FUNCTION_BLOCK FB_XPlanar_EM EXTENDS FB_PackML_BaseModule
VAR
    // Sub module definitions here

    // List of sub modules
    ipSubModules_Init : ARRAY[1..Parameters_PackML_Base.MAX_NO_OF_SUBMODULES] OF I_PackML_BaseModule := [];

    // Component definitions here
    XPlanarTable : FB_Component_Xplanar := (Name := 'XPlanarTable');
	
	//Station Components
	Station1	 : FB_DecisionStation	 := (Name := 'DecisionPoint');   //Declaration of a custom station
	Station2	 : FB_SpinStation 		 := (Name := 'RotateStation');
	Station3	 : FB_XPlanarStationBase := (Name := 'InspectStation');  //If no custom processing is needed simply declare an instance of the Station Base fb	 

    // List of Components
    ipComponents_Init : ARRAY[1..Parameters_PackML_Base.MAX_NO_OF_COMPONENTS] OF I_ComponentBase := [XPlanarTable, Station1, Station2, Station3];

    //Helper Vars
	Movers			  : ARRAY[1..Tc3_XPlanarStandard.Params_XPlanar.moverCount] OF FB_XPlanarMover;
	Tracks			  : ARRAY[1..Tc3_XPlanarStandard.Params_XPlanar.maxTrackCount] OF FB_XPlanarTrackSegment;
	
	
	fbinitbasic						: FB_BasicInitialization;
	aLocationOfArea 			: ARRAY[1..4,1..2] OF REAL:=[0,480,960,480,0,0,960,0];
	aManualPos					: ARRAY [1..19,1..2] OF REAL:=[60,420,240,420,420,420,600,420,860,420,60,300,240,300,420,300,600,300,860,300,60,180,240,180,420,180,600,180,860,180, 60,60,310,60,560,60,820,60];	
	
END_VAR

//! @summary This method contains code which will execute when this PackML module is in the <b>Aborting</b> state
METHOD PROTECTED Aborting
VAR
    i               : UDINT;
    SubModulesReady : BOOL := TRUE;
END_VAR

(*! <description> <b>Note:</b> The <i>Abort</i> command should be associated with the fault handing routine of a module. It should not be directly commanded from any user inteface. 

<table> 
	<tr>
		<th> Previous State </th>
		<th> Transition In </th>
		<th> Transition Out </th>
		<th> Next State  </th> 
	</tr>
	<tr>
		<td> <b>ANY</b> </td>
		<td> Abort Command </td> 
		<td> State Complete </td>
		<td> Aborted </td> 
	</tr>
</table>

This method is called as required by <c>StateControl()</c>
</description> 

*)
CASE DescendantSequenceState OF
    0:
        NoStateTasksToComplete  := FALSE;
        DescendantSequenceState := NextStep(DescendantSequenceState);

    10:
        IF XPlanarTable.Abort() THEN
            StateTasksComplete      := TRUE;
            DescendantSequenceState := NextStep(DescendantSequenceState);
        END_IF

    20:
        StateTasksComplete := TRUE;
END_CASE

SUPER^.Aborting();
END_METHOD

//! @summary This method contains code which will execute when this PackML module is in the <b>Clearing</b> state
METHOD PROTECTED Clearing
VAR
    i               : UDINT;
    SubModulesReady : BOOL := TRUE;
END_VAR

(*! <description> <b>Note:</b> The <i>Clear</i> command can also be thought of as a <i>fault reset</i> depite the ambiguity in the naming of the <i>Reset</i> state. 
<table> 
	<tr>
		<th> Previous State </th>
		<th> Transition In </th>
		<th> Transition Out </th>
		<th> Next State  </th> 
	</tr>
	<tr>
		<td> Aborted </td>
		<td> Clear Command </td> 
		<td> State Complete </td>
		<td> Stopped </td> 
	</tr>
</table>
This method is called as required by <c>StateControl()</c>
</description> 

*)
CASE _CurrentMode OF
    E_PMLUnitMode.ePMLUnitMode_Production:
        CASE DescendantSequenceState OF
            0: //Init
                NoStateTasksToComplete  := FALSE;
                XPlanarTable._Error     := FALSE;
				Station1.Reset();
				Station2.Reset();
				Station3.Reset();
			
                DescendantSequenceState := NextStep(DescendantSequenceState);

            10: //Check for Track initialization
                IF NOT XPlanarTable.TracksInitialized THEN
                    DescendantSequenceState := NextMinorStep(DescendantSequenceState);
                ELSE
                    DescendantSequenceState := NextStep(DescendantSequenceState);
                END_IF

            11: //Build Track Segments
                IF XPlanarTable.BuildTracks() THEN
                    IF NOT XPlanarTable.Error THEN
                      DescendantSequenceState := NextStep(DescendantSequenceState);
                    ELSE
                        DescendantSequenceState := 999;
                    END_IF;
                END_IF

            20: //Enable Group
                IF XPlanarTable.EnableGroup() THEN
                    DescendantSequenceState := NextStep(DescendantSequenceState);
                END_IF

            30:
                //Clearing complete
				fbinitbasic(bReset:=TRUE);
                StateTasksComplete := TRUE;
        END_CASE

    E_PMLUnitMode.ePMLUnitMode_Manual:
        ;
END_CASE

SUPER^.Clearing();
END_METHOD

METHOD PROTECTED CreateEvents
VAR_INPUT
END_VAR
// Add your event creation here

// Super call to base
SUPER^.CreateEvents();
END_METHOD

METHOD CyclicLogic
VAR
    i : INT;
    j : UDINT;
END_VAR
IF NOT _InitComplete THEN
    _InitComplete := Initialize();
END_IF

SUPER^.CyclicLogic();

IF _InitComplete THEN
	FOR j := 1 TO MAX_STATION_NUMBER DO
		stStationVis[j].bInit := TRUE;
		stStationVis[j].fPosition_X := stStationPos[j].fpositionX;		
		stStationVis[j].fPosition_Y := stStationPos[j].fpositionY;		
	END_FOR
	FOR j := 1 TO Tc3_XPlanarStandard.Params_XPlanar.moverCount DO
		stMoverVis[j].fPosition_X := Movers[j].std.P_ActPosition.x;		
		stMoverVis[j].fPosition_Y := Movers[j].std.P_ActPosition.y;	
		stMoverVis[j].fPosition_C := Movers[j].std.P_ActPosition.c;			
	END_FOR	
	

END_IF
END_METHOD

//! @summary This method contains code which will execute when this PackML module is in the <b>Execute</b> state
METHOD PROTECTED Execute
VAR
    i : UDINT;
END_VAR
VAR_INST
	InspectSimTimer: TON;
END_VAR
(*! <description> <b>The base implementation of this method is empty. User must override this method to provide functionality.</b>
<table> 
	<tr>
		<th> Previous State </th>
		<th> Transition In </th>
		<th> Transition Out </th>
		<th> Next State  </th> 
	</tr>
	<tr>
		<td> Starting<b>-or-</b>Unholding <b>-or-</b>Unsuspending</td>
		<td> State Complete<i>(Starting<b>-or-</b>Unholding<b>-or-</b>Unsuspending)</i></td> 
		<td> State Complete<b>-or-</b>Hold Command<b>-or-</b>Suspend Command</td>
		<td> Completing<b>-or-</b>Holding<b>-or-</b>Suspending</td>
	</tr>
</table>
This method is called as required by <c>StateControl()</c>
</description> 

*)
CASE _CurrentMode OF
    E_PMLUnitMode.ePMLUnitMode_Production:
        FOR i := 1 TO Params_XPlanar.maxNumStation DO
            ip.Stations[i].Execute();
        END_FOR
	
	//Simulate the "Inspection Done" signal
	InspectSimTimer(IN := ip.Stations[3].StationReady, PT := T#1S);
	ip.Stations[3].StationComplete := InspectSimTimer.Q;
	
    E_PMLUnitMode.ePMLUnitMode_Manual:
        ;
END_CASE
END_METHOD

//! @summary Automatically enables and disables HMI control based on the PackML mode
METHOD PROTECTED HMIPermissions

//! @description This method is called cyclically by <c>CyclicLogic()</c>
//General Mode Based Monitoring and handling of HMI control
CASE _CurrentMode OF
    E_PMLUnitMode.ePMLUnitMode_Production:
        AllowHMIControl(ThisModuleOnly := FALSE);

    E_PMLUnitMode.ePMLUnitMode_Manual:
        AllowHMIControl(ThisModuleOnly := FALSE);

    E_PMLUnitMode.ePMLUnitMode_Maintenance:
        AllowHMIControl(ThisModuleOnly := FALSE);
END_CASE
END_METHOD

//! @summary Basic module initialization logic
METHOD PROTECTED Initialize : BOOL;
VAR
    i                        : UDINT;
    varInfo                  : __SYSTEM.VAR_INFO;
    AllSubUnitsInitialized   : BOOL := TRUE;
    AllComponentsInitialized : BOOL := TRUE;
    tmpMoveDynamics          : ST_MoveDynamics;
    stHaltDynamics           : ST_HaltDynamics;
END_VAR

//! @description This method is called by <c>CyclicLogic()</c> as required
Initialize := FALSE;
CASE DescendantSequenceState OF
	0:
		// Define the interfaces to the different subunits (Must take place before SUPER^.initialize call)
		FOR i := 1 TO SPT_BaseTypes.Parameters_PackML_Base.MAX_NO_OF_SUBMODULES DO
			ipSubModules[i] := ipSubModules_Init[i];
		END_FOR

		FOR i := 1 TO SPT_BaseTypes.Parameters_PackML_Base.MAX_NO_OF_COMPONENTS DO
			ipComponents[i] := ipComponents_Init[i];
		END_FOR

		_LogModeChanges			:= FALSE;
		_LogStateChanges		:= FALSE;
		DescendantSequenceState := DescendantSequenceState + 10;

	10:
		//Set Mover and Track interfaces
		FOR i := 1 TO Tc3_XPlanarStandard.Params_XPlanar.moverCount DO
			Movers[i].MoverIndex := i;
			ip.Movers[i]		  := Movers[i];
		END_FOR

		FOR i := 1 TO Tc3_XPlanarStandard.Params_XPlanar.maxTrackCount DO
			ip.Tracks[i] := Tracks[i];
		END_FOR

		DescendantSequenceState := DescendantSequenceState + 10;

	20:
		//Copy Mode names
		FOR i := 1 TO 3 DO
			ModeNames[i] := F_UnitModeToString(UDINT_TO_DINT(i));
		END_FOR

		DescendantSequenceState := DescendantSequenceState + 10;

	30:
		//Call the Super
		IF SUPER^.Initialize() THEN
			DescendantSequenceState := DescendantSequenceState + 10;
		END_IF

	40:
		IF SetupTrackSegments() THEN
			DescendantSequenceState := DescendantSequenceState + 10;
		END_IF

	50:
		IF SetupStations() THEN
			DescendantSequenceState := DescendantSequenceState + 10;
		END_IF

	60:
		stHaltDynamics.PathXY.fVelocity		:= 500.0;
		stHaltDynamics.PathXY.fAcceleration := 10000.0;
		stHaltDynamics.PathXY.fDeceleration := 10000.0;
		stHaltDynamics.PathXY.fJerk			:= 100000.0;
		stHaltDynamics.AxisX.fVelocity		:= 500.0;
		stHaltDynamics.AxisX.fAcceleration	:= 10000.0;
		stHaltDynamics.AxisX.fDeceleration	:= 10000.0;
		stHaltDynamics.AxisX.fJerk			:= 100000.0;
		stHaltDynamics.AxisY.fVelocity		:= 500.0;
		stHaltDynamics.AxisY.fAcceleration	:= 10000.0;
		stHaltDynamics.AxisY.fDeceleration	:= 10000.0;
		stHaltDynamics.AxisY.fJerk			:= 100000.0;
		stHaltDynamics.AxisZ.fVelocity		:= 500.0;
		stHaltDynamics.AxisZ.fAcceleration	:= 10000.0;
		stHaltDynamics.AxisZ.fDeceleration	:= 10000.0;
		stHaltDynamics.AxisZ.fJerk			:= 100000.0;
		stHaltDynamics.AxisA.fVelocity		:= 10.0;
		stHaltDynamics.AxisA.fAcceleration	:= 100.0;
		stHaltDynamics.AxisA.fDeceleration	:= 100.0;
		stHaltDynamics.AxisA.fJerk			:= 100.0;
		stHaltDynamics.AxisB.fVelocity		:= 10.0;
		stHaltDynamics.AxisB.fAcceleration	:= 100.0;
		stHaltDynamics.AxisB.fDeceleration	:= 100.0;
		stHaltDynamics.AxisB.fJerk			:= 100.0;
		stHaltDynamics.AxisC.fVelocity		:= 36.0;
		stHaltDynamics.AxisC.fAcceleration	:= 360.0;
		stHaltDynamics.AxisC.fDeceleration	:= 360.0;
		stHaltDynamics.AxisC.fJerk			:= 360.0;
		FOR i := 1 TO Params_XPlanar.moverCount DO
			ip.Movers[i].std.P_HaltDynamics := stHaltDynamics;
		END_FOR

		Initialize := TRUE;
END_CASE
END_METHOD

//! @summary This method contains code which will execute when this PackML module is in the <b>Resetting</b> state
METHOD PROTECTED Resetting
VAR
	SubModulesReady : BOOL := TRUE;
END_VAR

VAR_INST
	i : UDINT;
END_VAR

(*! <description> <b>Note:</b> The <i>Reset</i> command can also be thought of as an <i>enable</i> depite the ambiguity in the naming of the <i>Clearing</i> state.
<table> 
	<tr>
		<th> Previous State </th>
		<th> Transition In </th>
		<th> Transition Out </th>
		<th> Next State  </th> 
	</tr>
	<tr>
		<td> Stopped<b>-or-</b>Completed </td>
		<td> Reset Command </td> 
		<td> State Complete </td>
		<td> Idle </td> 
	</tr>
</table>
This method is called as required by <c>StateControl()</c>
</description> 

*)
CASE _CurrentMode OF
	E_PMLUnitMode.ePMLUnitMode_Production:
		CASE DescendantSequenceState OF
			0: //Init
				i						:= 1;
				NoStateTasksToComplete	:= FALSE;
				DescendantSequenceState := NextStep(DescendantSequenceState);

			10: //Reset XPlanar System
				IF XPlanarTable.Reset() THEN
					DescendantSequenceState := NextStep(DescendantSequenceState);
				END_IF

			20: //Enable Tracks
				IF XplanarTable.EnableTracks(FALSE) THEN
					DescendantSequenceState := NextStep(DescendantSequenceState);
				END_IF

			30: //Enable Movers
				IF XPlanarTable.EnableMovers(FALSE) THEN
					DescendantSequenceState := NextStep(DescendantSequenceState);
				END_IF

			40: //Check Mover Angle
				IF i <= Params_XPlanar.moverCount THEN
					IF ip.Movers[1].SquareUp() THEN
						DescendantSequenceState := NextMinorStep(DescendantSequenceState);
					END_IF
				ELSE
					DescendantSequenceState := NextStep(DescendantSequenceState);
				END_IF
				
			41: //CheckMoverCount
				IF i <= Params_XPlanar.moverCount THEN
					i := i + 1;
					DescendantSequenceState := 40;
				ELSE
					DescendantSequenceState := NextStep(DescendantSequenceState);
				END_IF				

			50: //Clearing complete
				StateTasksComplete := TRUE;
		END_CASE
END_CASE

SUPER^.Resetting();
END_METHOD

METHOD PRIVATE SetupStations : BOOL
VAR_INPUT
END_VAR
stStationPos[1].fpositionX:=120;
stStationPos[1].fpositionY:=240;
stStationPos[2].fpositionX:=360;
stStationPos[2].fpositionY:=360;
stStationPos[3].fpositionX:=360;
stStationPos[3].fpositionY:=120;






//Set Required Process Station Initialization Parameters
Station1.Position.SetValuesXYC(stStationPos[1].fpositionX, stStationPos[1].fpositionY, 0);		 //Set the center of the station
Station1.TrackID	 := ip.Tracks[1];				 //Set the interface of the track segment the station resides on
Station1.StationType := E_StationType.DecisionPoint; //Change the type to Decision Point only if the station is acting as a divert and processing on the fly
Station1.OutputA	 := Station2;					 //Set any custom station parameters
Station1.OutputB	 := Station3;
ip.Stations[1]		 := Station1; 					 //Register the station with the interface array

Station2.Position.SetValuesXYC(stStationPos[2].fpositionX, stStationPos[2].fpositionY, 0);
Station2.Size.x		 := 120;						 //Changes the station size in the X plane
Station2.Size.y		 := 120; 						 //Changes the station size in the Y plane
Station2.TrackID	 := ip.Tracks[2];
Station2.NextStation := Station1; 					 //Set the interface for the next station of the mover
ip.Stations[2]		 := Station2;

Station3.Position.SetValuesXYC(stStationPos[3].fpositionX, stStationPos[3].fpositionY, 0);
Station3.Size.x		 := 120;
Station3.Size.y		 := 120;
Station3.TrackID	 := ip.Tracks[3];
Station3.NextStation := Station1;
ip.Stations[3]		 := Station3;
SetupStations		 := TRUE;
END_METHOD

METHOD PRIVATE SetupTrackSegments : BOOL
VAR_INST
    nSegmentIndex : UDINT;
END_VAR

VAR
    ResultAddPoint : INT;
END_VAR
SetupTrackSegments := FALSE;
CASE nSegmentIndex OF
	0: //Get ready
		nSegmentIndex := nSegmentIndex + 1;

	//********************************************************************************************************************************

	//Add states for each track segment in the system

	//********************************************************************************************************************************
	1:
		ip.Tracks[nSegmentIndex].ID := nSegmentIndex;
		IF ip.Tracks[nSegmentIndex].TrackTable.ClearTrackTable() THEN
			ResultAddPoint := ip.Tracks[nSegmentIndex].TrackTable.AddPoint(E_PointType.Line_Start,
																		   E_PointOption.none,
																		   300,//480.0,
																		   120,//20.0,
																		   0.0);

			ResultAddPoint := ip.Tracks[nSegmentIndex].TrackTable.AddPoint(E_PointType.Line_End,
																		   E_PointOption.none,
																		   130,//240.0,
																		   120,//120.0,
																		   0.0);

			ResultAddPoint := ip.Tracks[nSegmentIndex].TrackTable.AddPoint(E_PointType.Line_Start,
																		   E_PointOption.none,
																		   120,//20.0,
																		   130,//240.0,
																		   0.0);

			ResultAddPoint := ip.Tracks[nSegmentIndex].TrackTable.AddPoint(E_PointType.Line_End,
																		   E_PointOption.none,
																		   120,//120.0,
																		   240,//480.0,
																		   0.0);

//			ResultAddPoint := ip.Tracks[nSegmentIndex].TrackTable.AddPoint(E_PointType.Line_Start,
//																		   E_PointOption.none,
//																		   120,//240.0,
//																		   300,//600.0,
//																		   0.0);

//			ResultAddPoint := ip.Tracks[nSegmentIndex].TrackTable.AddPoint(E_PointType.Line_End,
//																		   E_PointOption.none,
//																		   240,//480.0,
//																		   300,//600.0,
//																		   0.0);

			ip.Tracks[nSegmentIndex].TrackTable.P_CloseTheLoop := FALSE;
		END_IF

		nSegmentIndex := nSegmentIndex + 1;

	2:
		ip.Tracks[2].ID := 2;  															//Set the ID property of the track segment
		IF ip.Tracks[2].TrackTable.ClearTrackTable() THEN								//Clean up any stray points in the table
			ResultAddPoint := ip.Tracks[2].TrackTable.AddPoint(E_PointType.Line_Start,	//Configure track points
															   E_PointOption.none,
															   120,//600.0,
															   240,//480.0,
															   0.0);

			ResultAddPoint := ip.Tracks[2].TrackTable.AddPoint(E_PointType.Line_End,
															   E_PointOption.none,
															   120,//600.0,
															   350,//240.0,
															   0.0);
															   
			ResultAddPoint := ip.Tracks[2].TrackTable.AddPoint(E_PointType.Line_Start,	//Configure track points
															   E_PointOption.none,
															   130,//600.0,
															   360,//480.0,
															   0.0);

			ResultAddPoint := ip.Tracks[2].TrackTable.AddPoint(E_PointType.Line_End,
															   E_PointOption.none,
															   360,//600.0,
															   360,//240.0,
															   0.0);			

			ResultAddPoint := ip.Tracks[2].TrackTable.AddPoint(E_PointType.Line_Start,	//Configure track points
															   E_PointOption.none,
															   360,//600.0,
															   330,//480.0,
															   0.0);

			ResultAddPoint := ip.Tracks[2].TrackTable.AddPoint(E_PointType.Line_End,
															   E_PointOption.none,
															   360,//600.0,
															   240,//240.0,
															   0.0);											   

			ip.Tracks[2].TrackTable.P_CloseTheLoop	 := FALSE;						//Set the segment close the loop property		
			ip.Tracks[2].TrackTable.P_StartFromTrack := ip.Tracks[1].std;			//If linking to a previous track segment set the interface
			ip.Tracks[2].TrackTable.P_EndAtTrack	 := ip.Tracks[1].std;			//If linking to a downstream track segment set the interface
		END_IF

		nSegmentIndex := nSegmentIndex + 1;

	3:
		ip.Tracks[nSegmentIndex].ID := nSegmentIndex;
		IF ip.Tracks[nSegmentIndex].TrackTable.ClearTrackTable() THEN
			ResultAddPoint := ip.Tracks[nSegmentIndex].TrackTable.AddPoint(E_PointType.Line_Start,
																		   E_PointOption.none,
																		   140,//480.0,
																		   240,//600.0,
																		   0.0);

			ResultAddPoint := ip.Tracks[nSegmentIndex].TrackTable.AddPoint(E_PointType.Line_End,
																		   E_PointOption.none,
																		   350,//720.0,
																		   240,//600.0,
																		   0.0);

			ResultAddPoint := ip.Tracks[nSegmentIndex].TrackTable.AddPoint(E_PointType.Line_Start,
																		   E_PointOption.none,
																		   360,//840.0,
																		   230,//480.0,
																		   0.0);

			ResultAddPoint := ip.Tracks[nSegmentIndex].TrackTable.AddPoint(E_PointType.Line_End,
																		   E_PointOption.none,
																		   360,//840.0,
																		   120,//240.0,
																		   0.0);

//			ResultAddPoint := ip.Tracks[nSegmentIndex].TrackTable.AddPoint(E_PointType.Line_Start,
//																		   E_PointOption.none,
//																		   360,//720.0,
//																		   60,//120.0,
//																		   0.0);

//			ResultAddPoint := ip.Tracks[nSegmentIndex].TrackTable.AddPoint(E_PointType.Line_End,
//																		   E_PointOption.none,
//																		  240,// 480.0,
//																		   60,//120.0,
//																		   0.0);

			ip.Tracks[nSegmentIndex].TrackTable.P_CloseTheLoop	 := FALSE;
			ip.Tracks[nSegmentIndex].TrackTable.P_StartFromTrack := ip.Tracks[1].std;
			ip.Tracks[nSegmentIndex].TrackTable.P_EndAtTrack	 := ip.Tracks[1].std;
		END_IF

		nSegmentIndex := nSegmentIndex + 1;
		
	4:
		ip.Tracks[nSegmentIndex].ID := nSegmentIndex;
		IF ip.Tracks[nSegmentIndex].TrackTable.ClearTrackTable() THEN
			ResultAddPoint := ip.Tracks[nSegmentIndex].TrackTable.AddPoint(E_PointType.Line_Start,
																		   E_PointOption.none,
																		   60,//100.0,
																		   420,//100.0,
																		   0.0);

			ResultAddPoint := ip.Tracks[nSegmentIndex].TrackTable.AddPoint(E_PointType.Line_End,
																		   E_PointOption.none,
																		   420,//100.0,
																		   420,//500.0,
																		   0.0);

			ResultAddPoint := ip.Tracks[nSegmentIndex].TrackTable.AddPoint(E_PointType.Line_Start,
																		   E_PointOption.none,
																		   420,//240.0,
																		   300,//620.0,
																		   0.0);

			ResultAddPoint := ip.Tracks[nSegmentIndex].TrackTable.AddPoint(E_PointType.Line_End,
																		   E_PointOption.none,
																		   60,//780.0,
																		   300,//620.0,
																		   0.0);

			ResultAddPoint := ip.Tracks[nSegmentIndex].TrackTable.AddPoint(E_PointType.Line_Start,
																		   E_PointOption.none,
																		   60,//860.0,
																		   180,//480.0,
																		   0.0);

			ResultAddPoint := ip.Tracks[nSegmentIndex].TrackTable.AddPoint(E_PointType.Line_End,
																		   E_PointOption.none,
																		   420,//860.0,
																		   180,//240.0,
																		   0.0);
																		   
			ResultAddPoint := ip.Tracks[nSegmentIndex].TrackTable.AddPoint(E_PointType.Line_Start,
																		   E_PointOption.none,
																		   420,//860.0,
																		   60,//240.0,
																		   0.0);					

			ResultAddPoint := ip.Tracks[nSegmentIndex].TrackTable.AddPoint(E_PointType.Line_End,
																		   E_PointOption.none,
																		   60,//860.0,
																		   60,//240.0,
																		   0.0);													

			ip.Tracks[nSegmentIndex].TrackTable.P_CloseTheLoop	 := FALSE;
			ip.Tracks[nSegmentIndex].TrackTable.P_EndAtTrack	 := ip.Tracks[1].std;
		END_IF

		nSegmentIndex := nSegmentIndex + 1;		

	5:
		nSegmentIndex	   := 0;
		SetupTrackSegments := TRUE;
END_CASE
END_METHOD

//! @summary This method contains code which will execute when this PackML module is in the <b>Starting</b> state
METHOD PROTECTED Starting
VAR
    SubModulesReady : BOOL := TRUE;
    Position        : PositionXYC;
    check           : ST_CheckStartConditionFeedback;
    lError          : BOOL;
    lErrorID        : UDINT;
    Angle           : LREAL;
END_VAR

VAR_INST
    MoverNumber       : UDINT;
    StationNumber     : UDINT;
    ipMover           : ARRAY [0..Tc3_XPlanarStandard.Params_XPlanar.moverCount] OF I_XPlanarMover;
    ipStation         : I_XPlanarStation;
    JoinState         : INT;
    MoveState         : INT;
    i                 : UDINT;
    JoinTrackNum      : UINT;
    MoveStationNum    : ARRAY[1..Params_XPlanar.moverCount] OF UINT;
    MoveStationNeeded : ARRAY[1..Params_XPlanar.moverCount] OF BOOL;
    JoinStationNeeded : ARRAY[1..Params_XPlanar.moverCount] OF BOOL;
END_VAR
CASE _CurrentMode OF
	E_PMLUnitMode.ePMLUnitMode_Production:
		CASE DescendantSequenceState OF
			0:
				NoStateTasksToComplete	:= FALSE;
				DescendantSequenceState := 10;
				StationNumber			:= 1;
				i						:= 1;
				JoinState				:= 0;

			10: //Clean Up Mover Queues
				FOR i := 1 TO Params_XPlanar.moverCount DO
					ip.Movers[i].Destination := 0;
				END_FOR

				FOR i := 1 TO Params_XPlanar.maxNumStation DO
					ip.Stations[i].MoverQueue.Dequeue();
				END_FOR

				i						:= 1;
				DescendantSequenceState := 15;
//				DescendantSequenceState := NextStep(DescendantSequenceState);
				
			15:
				fbinitbasic(bExcute:=TRUE,nSizeOfMover:=115,aLocationOfArea:=aLocationOfArea,ipMover:=ip.Movers,aManualPos:=aManualPos,bReset:=);
				IF fbinitbasic.Done THEN
//						DescendantSequenceState := NextStep(DescendantSequenceState);		
				END_IF
			

			20: //Join Movers to recovery track
				IF i <= Params_XPlanar.moverCount THEN
					IF ip.Movers[i].JoinTrack(ip.Tracks[4]) THEN
						DescendantSequenceState := NextMinorStep(DescendantSequenceState);
					END_IF
				ELSE
					i						:= 1;
					DescendantSequenceState := NextStep(DescendantSequenceState);
				END_IF
				
			21: //Check Mover Count
				IF i <= Params_XPlanar.moverCount THEN
 					i := i + 1;
					DescendantSequenceState := 20;
				ELSE
					i						:= 1;
					DescendantSequenceState := NextStep(DescendantSequenceState);
				END_IF					

			30: //Send Movers around to station 1
				IF i <= Params_XPlanar.moverCount THEN
					IF ip.Movers[i].SendToStation(ip.Stations[1]) THEN
						DescendantSequenceState := NextMinorStep(DescendantSequenceState);
					END_IF
				ELSE
					i						:= 1;
					DescendantSequenceState := NextStep(DescendantSequenceState);
				END_IF
				
			31: //Check Mover Count
				IF i <= Params_XPlanar.moverCount THEN
 					i := i + 1;
					DescendantSequenceState := 30;
				ELSE
					i						:= 1;
					DescendantSequenceState := NextStep(DescendantSequenceState);
				END_IF	

			40:
				StateTasksComplete := TRUE;
		END_CASE

	E_PMLUnitMode.ePMLUnitMode_Manual:
		;
END_CASE

SUPER^.Starting();
END_METHOD

END_FUNCTION_BLOCK

(* stored: Version 1.1.0.1, ProductVersion 3.1.4024.12
   POU FB_XPlanar_EM: Id {18ed3aa7-c83f-44ce-8119-20fe14cb0cfa}, SpecialFunc None
   Folder I_CyclicFB: Id {769d746d-1ab5-4a6d-8c77-4b1403733257}
   Folder Methods: Id {1414b749-8a1b-4539-8751-a9eb98ce9efa}
   Folder Acting States: Id {f6cfc130-33f5-4b9c-9ed3-b6e57724e54f}
   Folder HMI: Id {0f08a4f8-e768-454b-a528-0661effe207e}
   Folder Waiting States: Id {ab86d3ba-50da-471d-864b-21041ca20d53}
   Method Aborting: Id {17e4bd4f-b401-48a2-abdb-1c82c9b91958}
   Method Clearing: Id {749d9d49-762f-4674-b533-d711fd25e786}
   Method CreateEvents: Id {72c60c54-f456-4c10-a113-470233e3942b}
   Method CyclicLogic: Id {31fa8ff0-2b84-4416-a54a-15ba032d89ac}
   Method Execute: Id {4a8447c7-4bba-456b-ae99-02b9655bd430}
   Method HMIPermissions: Id {7d2cddec-eedc-414c-8c02-c97cb122267e}
   Method Initialize: Id {cea669eb-9427-49e9-a099-b64514cc633b}
   Method Resetting: Id {31624805-9f24-4846-bb15-1edf775cd7f4}
   Method SetupStations: Id {472d87c4-f8ee-4679-a5bf-c6f2e3004197}
   Method SetupTrackSegments: Id {c993939d-20e4-4cee-b613-07c22d3b3260}
   Method Starting: Id {183f1123-c447-4a86-b202-a4cab71a6c14} *)
